# EPICS substitutions: ek9000App/Db/EL1144_mbbiDirect.substitutions
file EL1144.template
{       pattern
        {
                TERMINAL,

        }
        {
        }
}
